// TwinCAT 3 PLC project log4Tc_Tester
// ProgramVersion: 3.1.4026.20
// CompilerDefines: DEBUG
// libraries:
//   Log4TC, * (mbc engineering GmbH)
//   Tc2_Standard, * (Beckhoff Automation GmbH)
//   Tc2_System, * (Beckhoff Automation GmbH)
//   Tc2_Utilities, * (Beckhoff Automation GmbH)
//   Tc3_Module, * (Beckhoff Automation GmbH)
//   Base Interfaces,newest,System
// project tree:
//   GVLs/ GVL.TcGVL (not stored)
//   / PlcTask.TcTTO (not stored)
//   POUs/ CheckBounds.TcPOU (not stored), CheckLRangeSigned.TcPOU (not stored), CheckLRangeUnsigned.TcPOU (not stored), CheckPointer.TcPOU (not stored), CheckRangeSigned.TcPOU (not stored), CheckRangeUnsigned.TcPOU (not stored), FB_TcExternalTime.TcPOU (not stored), F_FUN.TcPOU (not stored) (excluded from build), MAIN.TcPOU (not stored), PRG_TestSimpleApi.TcPOU
// (motion and I/O tree: see PLC project log4tc)
// real-time tasks:
//   TASK PlcTask: cycle T#1ms, priority 20, ADS port 350
//   TASK PlcTask1: cycle T#10ms, priority 21, ADS port 351

// ---- POUs/PRG_TestSimpleApi.TcPOU
PROGRAM PRG_TestSimpleApi
VAR
	bExecute		: BOOL;
	bExecuteSingle	: BOOL;
	
	nArg			: INT := 42;
	sArg			: T_MaxString := 'foo';
	fArg			: REAL := 4.2;
	
	tTime			: TIME :=  T#12H34M15S;
	tLTime			: LTIME := LTIME#1000D15H23M12S34MS2US44NS;
	dDate			: DATE := DATE#1996-05-06;
	dDT				: DT := DATE_AND_TIME#1996-05-06-15:36:30;
	tTOD			: TOD := TIME_OF_DAY#15:36:30.123;
	eEnum			: E_LogLevel := E_LogLevel.eFatal;
	wStr			: WSTRING := "fooöäaΘ𝄞";
	
	fbScope			: FB_ScopedContext;
END_VAR

//fbScope.ContextBuilder.AddInt('scope', 42);

IF bExecute OR bExecuteSingle THEN
	bExecuteSingle := FALSE;

// 	F_LogLA1C(
// 		E_LogLevel.eInfo, 
// 		'PRG_TestSimpleApi', 
// 		'Temperatur {temperature}', 
// 		fArg, 
// 		//F_LogContext().AddBool('csv', TRUE)
// 	);
	
	
	F_LogA7(
		E_LogLevel.eInfo, 
		'Neue Datentypen TIME={time} LTIME={ltime} DATE={date} DT={date_and_time} TOD={time_of_day} ENUM={enum} WSTRING={wstring}',
		tTime,
		tLTime,
		dDate,
		dDT,
		tTOD,
		eEnum,
		wStr
	);
		
		
	
	(*
	
	fbScope.Begin();
	
	F_LogLA3(
		E_LogLevel.eInfo,
		'PRG_TestSimpleApi',
		'Log F_LogLA3({arg1},{arg2},{arg3})',
		nArg,
		sArg,
		fArg,
	);
	
	fbScope.End();
	
	F_LogA3(
		E_LogLevel.eInfo,
		'Log F_LogA3({arg1},{arg2},{arg3})',
		nArg,
		sArg,
		fArg
	);
	¨*)
	
END_IF

END_PROGRAM
